Fanuc TP program (LS listing): p_m45.ls

/PROG  P_M45
/ATTR
OWNER		= MNEDITOR;
COMMENT		= "";
PROG_SIZE	= 508;
CREATE		= DATE 25-11-25  TIME 14:36:16;
MODIFIED	= DATE 25-12-17  TIME 16:06:24;
FILE_NAME	= P_45;
VERSION		= 0;
LINE_COUNT	= 1;
MEMORY_SIZE	= 876;
PROTECT		= READ_WRITE;
TCD:  STACK_SIZE	= 0,
      TASK_PRIORITY	= 50,
      TIME_SLICE	= 0,
      BUSY_LAMP_OFF	= 0,
      ABORT_REQUEST	= 0,
      PAUSE_REQUEST	= 0;
DEFAULT_GROUP	= *,1,*,*,*;
CONTROL_CODE	= 00000000 00000000;
LOCAL_REGISTERS	= 0,0,0;
/APPL
  ARC Welding Equipment : 1,*,*,*,*;

MPAS ;
MPAS_NUM_PASSES        : 0;
MPAS_LAST_PASS         : 0;
MPAS_CURRENT_PASS      : 0;
MPAS_STATUS_PASS       : 0;
/MN
   1:J P[1] 50% FINE    ;
/POS
P[1]{
   GP2:
	UF : 9, UT : 2,
	J1=   -45.000 deg
};
/END
